// TIA Portal V16 export
// export: Created 2021-11-12T13:31:53.8851244Z, ExportSetting WithDefaults, DisplayName Totally Integrated Automation Portal, DisplayVersion V16 Update 3, DisplayName TIA Portal Version Control Interface, DisplayVersion V16 Update 2, DisplayName TIA Portal Openness, DisplayVersion V16 Update 3, DisplayName SINAMICS Startdrive Advanced, DisplayVersion V16 Update 5, DisplayName SINAMICS Startdrive G130, G150, S120, S150, SINAMICS MV, S210, DisplayVersion V16 Update 5, DisplayName SINAMICS Startdrive G110M, G120, G120C, G120D, G120P, G115D, DisplayVersion V16 Update 5, DisplayName STEP 7 Professional, DisplayVersion V16 Update 3, DisplayName STEP 7 Safety, DisplayVersion V16, DisplayName WinCC UA Professional, DisplayVersion V16 Update 3
DATA_BLOCK "HMI_PARAM_MEM1"   // DB179
{ S7_Optimized_Access := 'TRUE' }
VERSION : 0.1
// stored: AutoNumber true, DBAccessibleFromOPCUA true, IsOnlyStoredInLoadMemory false, IsRetainMemResEnabled false, IsWriteProtectedInAS false, MemoryReserve 100
   VAR
      xxxxx___BinarySensors___xxxxx : Byte;
      xxxxx___Drives___xxxxx : Byte;
      xxxxx__Alarms__xxxxx { S7_SetPoint := 'True'} : Byte;
      MEM : "UDT_DI_Mon_Parameter";   // from MEM1
      LiveBit : "UDT_DI_Mon_Parameter";   // communication fault
      xxxxx__ProcesAlarms__xxxxx : Byte;
      xxxxx__SafetyAlarms__xxxxx : Byte;
   END_VAR
BEGIN
END_DATA_BLOCK
